(* IEC 61131-3 sources: json/test/Numbers, 6 files *)

(* ---- ItemTestDint.st ---- *)
USING AxUnit.Assert;
USING System.Strings;

NAMESPACE Simatic.Ax.Json
    {TestFixture}
    CLASS TestJsonElementsDint

        VAR PROTECTED
            e : JsonDInt := (Value := 999, Key := 'test');
            e2 : JsonDInt := (Value := -999, Key := 'second_key');
        END_VAR

        {Test}
        METHOD PUBLIC Test_Tostring_with_999_expect_test_999
            VAR_TEMP
                _str : STRING;
            END_VAR
            _str := e.ToString();
            Equal(expected := _str, actual := '"test": 999');
        END_METHOD

        {Test}
        METHOD PUBLIC Test_Tostring_with_Minus_999_expect_test_Minus_999
            Equal(expected := e2.ToString(), actual := '"second_key": -999');
        END_METHOD

    END_CLASS
END_NAMESPACE

(* ---- ItemTestInt.st ---- *)
USING AxUnit.Assert;
USING System.Strings;
USING Simatic.Ax.Conversion;

NAMESPACE Simatic.Ax.Json
    {TestFixture}
    CLASS TestJsonElementsInt

        VAR PROTECTED
            e : JsonInt := (Value := 999, Key := 'test');
            e2 : JsonInt := (Value := -999, Key := 'second_key');
            s_test_999 : STRING := '"test": 999';
            s_test_minus_999 : STRING := '"second_key": -999';
            cmpBuff : ARRAY[0..20] OF CHAR;
            doc : JsonDocument;
        END_VAR

        {Test}
        METHOD PUBLIC Test_Tostring_with_999_expect_test_999
            VAR_TEMP
                _str : STRING;
            END_VAR
            _str := e.ToString();
            Equal(expected := _str, actual := s_test_999);
        END_METHOD

        {Test}
        METHOD PUBLIC Test_Tostring_with_Minus_999_expect_test_Minus_999
            Equal(expected := e2.ToString(), actual := s_test_minus_999);
        END_METHOD

        {Test}
        METHOD PUBLIC TestSerialize_s_test_999
            VAR_TEMP
                len : DINT;
                res : BOOL;
            END_VAR
            e.Serialize(REF(doc));

            len := Strings.ToArray(str := s_test_999, arr := cmpBuff);
            res := CompareArray(first := doc.buffer, scnd := cmpBuff, count := TO_INT(len));
            Equal(expected := TRUE, actual := res);

        END_METHOD

        {Test}
        METHOD PUBLIC TestSerialize_s_test_minus_999
            VAR_TEMP
                len : DINT;
                res : BOOL;
            END_VAR

            e2.Serialize(REF(doc));
            len := Strings.ToArray(str := s_test_minus_999, arr := cmpBuff);
            res := CompareArray(first := doc.buffer, scnd := cmpBuff, count := TO_INT(len));
            Equal(expected := TRUE, actual := res);

        END_METHOD
    END_CLASS
END_NAMESPACE

(* ---- ItemTestSint.st ---- *)
USING AxUnit.Assert;
USING System.Strings;
USING Simatic.Ax.Conversion;

NAMESPACE Simatic.Ax.Json
    {TestFixture}
    CLASS TestJsonElementsSInt

        VAR PROTECTED
            e : JsonSInt := (Value := SINT#127, Key := 'test');
            e2 : JsonSInt := (Value := SINT#-128, Key := 'second_key');
            s_test_max : STRING := '"test": 127';
            s_test_min : STRING := '"second_key": -128';
            cmpBuff : ARRAY[0..20] OF CHAR;
            doc : JsonDocument;
            buffer : ARRAY[0..200] OF CHAR;
        END_VAR

        {Test}
        METHOD PUBLIC Test_Tostring_with_max_expect_test_max
            VAR_TEMP
                _str : STRING;
            END_VAR
            _str := e.ToString();
            Equal(expected := _str, actual := s_test_max);
        END_METHOD

        {Test}
        METHOD PUBLIC Test_Tostring_with_min_expect_test_min
            Equal(expected := e2.ToString(), actual := s_test_min);
        END_METHOD

        {Test}
        METHOD PUBLIC TestSerialize_s_test_max
            VAR_TEMP
                len : DINT;
                res : BOOL;
            END_VAR
            doc.buffer := REF(buffer);
            e.Serialize(REF(doc));

            len := Strings.ToArray.OfCharCount(str := s_test_max, arr := cmpBuff);
            res := CompareArray(first := buffer, scnd := cmpBuff, count := TO_INT(len));
            Equal(expected := TRUE, actual := res);

        END_METHOD

        {Test}
        METHOD PUBLIC TestSerialize_s_test_min
            VAR_TEMP
                len : DINT;
                res : BOOL;
            END_VAR
            doc.buffer := REF(buffer);
            e2.Serialize(REF(doc));
            len := Strings.ToArray.OfCharCount(str := s_test_min, arr := cmpBuff);
            res := CompareArray(first := buffer, scnd := cmpBuff, count := TO_INT(len));
            Equal(expected := TRUE, actual := res);

        END_METHOD
    END_CLASS
END_NAMESPACE

(* ---- ItemTestUInt.st ---- *)
USING AxUnit.Assert;
USING System.Strings;
USING Simatic.Ax.Conversion;

NAMESPACE Simatic.Ax.Json
    {TestFixture}
    CLASS TestJsonElementsUInt

        VAR PROTECTED
            e : JsonUInt := (Value := UINT#0, Key := 'test');
            e2 : JsonUInt := (Value := UINT#65535, Key := 'second_key');
            s_test_min : STRING := '"test": 0';
            s_test_max : STRING := '"second_key": 65535';
            cmpBuff : ARRAY[0..20] OF CHAR;
            doc : JsonDocument;
            buffer : ARRAY[0..200] OF CHAR;
        END_VAR

        {Test}
        METHOD PUBLIC Test_Tostring_with_min_expect_test_min
            VAR_TEMP
                _str : STRING;
            END_VAR
            _str := e.ToString();
            Equal(expected := _str, actual := s_test_min);
        END_METHOD

        {Test}
        METHOD PUBLIC Test_Tostring_with_max_expect_test_max
            Equal(expected := e2.ToString(), actual := s_test_max);
        END_METHOD

        {Test}
        METHOD PUBLIC TestSerialize_s_test_max
            VAR_TEMP
                len : DINT;
                res : BOOL;
            END_VAR
            doc.buffer := REF(buffer);
            e.Serialize(REF(doc));

            len := Strings.ToArray.OfCharCount(str := s_test_min, arr := cmpBuff);
            res := CompareArray(first := buffer, scnd := cmpBuff, count := TO_INT(len));
            Equal(expected := TRUE, actual := res);

        END_METHOD

        {Test}
        METHOD PUBLIC TestSerialize_s_test_min
            VAR_TEMP
                len : DINT;
                res : BOOL;
            END_VAR
            doc.buffer := REF(buffer);
            e2.Serialize(REF(doc));
            len := Strings.ToArray.OfCharCount(str := s_test_max, arr := cmpBuff);
            res := CompareArray(first := buffer, scnd := cmpBuff, count := TO_INT(len));
            Equal(expected := TRUE, actual := res);

        END_METHOD
    END_CLASS
END_NAMESPACE

(* ---- ItemTestUSint.st ---- *)
USING AxUnit.Assert;
USING System.Strings;
USING Simatic.Ax.Conversion;

NAMESPACE Simatic.Ax.Json
    {TestFixture}
    CLASS TestJsonElementsUSInt

        VAR PROTECTED
            e : JsonUSInt := (Value := USINT#255, Key := 'test');
            e2 : JsonUSInt := (Value := USINT#0, Key := 'second_key');
            s_test_max : STRING := '"test": 255';
            s_test_minus_min : STRING := '"second_key": 0';
            cmpBuff : ARRAY[0..20] OF CHAR;
            doc : JsonDocument;
        END_VAR

        {Test}
        METHOD PUBLIC Test_Tostring_with_999_expect_test_999
            VAR_TEMP
                _str : STRING;
            END_VAR
            _str := e.ToString();
            Equal(expected := _str, actual := s_test_max);
        END_METHOD

        {Test}
        METHOD PUBLIC Test_Tostring_with_Minus_999_expect_test_Minus_999
            Equal(expected := e2.ToString(), actual := s_test_minus_min);
        END_METHOD

        {Test}
        METHOD PUBLIC TestSerialize_s_test_999
            VAR_TEMP
                len : DINT;
                res : BOOL;
            END_VAR
            e.Serialize(REF(doc));

            len := Strings.ToArray.OfCharCount(str := s_test_max, arr := cmpBuff);
            res := CompareArray(first := doc.buffer, scnd := cmpBuff, count := TO_INT(len));
            Equal(expected := TRUE, actual := res);

        END_METHOD

        {Test}
        METHOD PUBLIC TestSerialize_s_test_minus_999
            VAR_TEMP
                len : DINT;
                res : BOOL;
            END_VAR

            e2.Serialize(REF(doc));
            len := Strings.ToArray.OfCharCount(str := s_test_minus_min, arr := cmpBuff);
            res := CompareArray(first := doc.buffer, scnd := cmpBuff, count := TO_INT(len));
            Equal(expected := TRUE, actual := res);

        END_METHOD
    END_CLASS
END_NAMESPACE

(* ---- TestJsonBoolean.st ---- *)
USING AxUnit.Assert;
USING System.Strings;
USING Simatic.Ax.Conversion;

NAMESPACE Simatic.Ax.Json
    {TestFixture}
    CLASS TestJsonBoolean

        VAR PROTECTED
            e : JsonBoolean := (Value := true, Key := 'test');
            e2 : JsonBoolean := (Value := false, Key := 'second_key');
            expString, actString : STRING;
            cmpBuff : ARRAY[0..20] OF CHAR;
            doc : JsonDocument;
        END_VAR

        {Test}
        METHOD PUBLIC TestSerialize_s_test_true
            VAR_TEMP
                len : DINT;
                res : BOOL;
            END_VAR
            e.Serialize(REF(doc));

            expString := '"test": true';
            len := Strings.ToArray(str := expString, arr := cmpBuff);
            res := CompareArray(first := doc.buffer, scnd := cmpBuff, count := TO_INT(len));
            Equal(expected := TRUE, actual := res);

        END_METHOD

        {Test}
        METHOD PUBLIC TestSerialize_s_test_minus_false
            VAR_TEMP
                len : DINT;
                res : BOOL;
            END_VAR

            e2.Serialize(REF(doc));
            expString := '"second_key": false';
            len := Strings.ToArray(str := expString, arr := cmpBuff);
            res := CompareArray(first := doc.buffer, scnd := cmpBuff, count := TO_INT(len));
            Equal(expected := TRUE, actual := res);

        END_METHOD
    END_CLASS
END_NAMESPACE
